// TwinCAT 3 PLC project
// project tree:
//   DUTs/ E_Error.TcDUT, ST_MyStruct.TcDUT, T_ALIAS.TcDUT
//   POUs/ F_SyntaxError.TcPOU, FB_MyBlock.TcPOU, FB_SecondBlock.TcPOU, MAIN.TcPOU, PlainFunction.TcPOU, PlainFunctionBlock.TcPOU, RegularFunction.TcPOU

// ---- DUTs/E_Error.TcDUT
{attribute 'qualified_only'}
{attribute 'strict'}
TYPE E_Error :
(
	OK := 0,
    SomeError := 5,
    OtherError
) USINT;
END_TYPE

// ---- DUTs/ST_MyStruct.TcDUT
TYPE ST_MyStruct :
STRUCT
    number      : LREAL;
    text        : STRING(10);
END_STRUCT
END_TYPE

// ---- DUTs/T_ALIAS.TcDUT
TYPE T_ALIAS : WORD;
END_TYPE

// ---- POUs/F_SyntaxError.TcPOU
FUNCTION F_SyntaxError RETURNS BOOL
VAR_INPUT
END_VAR

END_FUNCTION

// ---- POUs/FB_MyBlock.TcPOU
(*
Info!
*)
FUNCTION_BLOCK FB_MyBlock
VAR_INPUT
    someInput       : LREAL;        // This is some input with a description
    otherInput      : BOOL;         // Awesome description 
END_VAR
VAR_INPUT
    secondClause    : LREAL;        // This is some input with a description 
END_VAR
VAR_OUTPUT
    myOutput        : UINT;         // Return something nice
END_VAR
VAR
END_VAR

myOutput := 420;

METHOD AnotherMethod : LREAL
VAR_INPUT
    methodInput     : LREAL;            // Some input
END_VAR
END_METHOD

(*
This is a description.
*)
METHOD MyMethod : BOOL
VAR_INPUT
END_VAR
MyMethod := FALSE;
END_METHOD

END_FUNCTION_BLOCK

// ---- POUs/FB_SecondBlock.TcPOU
FUNCTION_BLOCK FB_SecondBlock EXTENDS FB_MyBlock
VAR_INPUT
END_VAR
VAR_OUTPUT
END_VAR
VAR
END_VAR

END_FUNCTION_BLOCK

// ---- POUs/MAIN.TcPOU
PROGRAM MAIN
VAR
    request         : UDINT := 0;
    ack             : UDINT := 0;
    
    block           : FB_MyBlock;
    
    result          : LREAL;
    
END_VAR

IF ack <> request THEN
    ack := request;
END_IF

result := RegularFunction(input := 3.14, other_arg := 7);

END_PROGRAM

// ---- POUs/RegularFunction.TcPOU
(*
Short description of the function.

Long description of the function, spanning multiple
rows even.
*)
FUNCTION RegularFunction : LREAL
VAR_INPUT
    input       : LREAL;            // This is an in-code description of some variable
    other_arg   : UDINT;
END_VAR
VAR
END_VAR

RegularFunction := input * 2.0;

END_FUNCTION

// ---- POUs/PlainFunction.TcPOU
FUNCTION PlainFunction : BOOL
VAR_INPUT
END_VAR
VAR
END_VAR

END_FUNCTION

// ---- POUs/PlainFunctionBlock.TcPOU
FUNCTION_BLOCK PlainFunctionBlock
VAR_INPUT
    someInput       : BOOL;
END_VAR
VAR_OUTPUT
    someOutput      : BOOL;
END_VAR
VAR
END_VAR

END_FUNCTION_BLOCK
